Fanuc KAREL source: kb00190.KL

-- PROVISIONAL review KL for V1013-1; original PC SHA256 701228a5c5395698bf2e7cdfde362432b9e381be210ff0e65e3f8c48e836c0e9
-- Incomplete behavior may be omitted. Consult companion uncertainty JSON. Do not deploy.
PROGRAM KB00190
%NOLOCKGROUP
VAR
  P1 : REAL
  RESULT : REAL
BEGIN
  -- UNRESOLVED_PC offsets 5-16; opcodes 2E,23
  -- UNRESOLVED_PC offsets 21-36; opcodes 27,22,76,23
  -- UNRESOLVED_PC offsets 41-45; opcodes 7F
END KB00190
